// Mitsubishi GX Works2 project: TIMMERs   PLC: Q03UDV

PROGRAM MAIN
VAR
  TS0 : BOOL;
  RT0 : BOOL;
  TMR1 : BOOL;
END_VAR
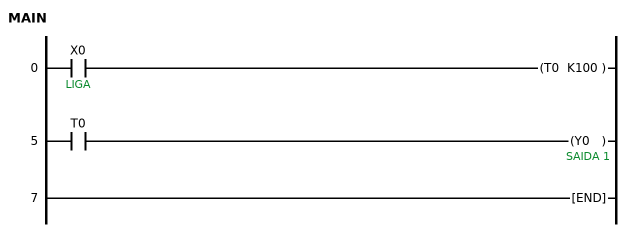
0     LD      X0  ; LIGA
      OUT     T0 K100
5     LD      T0
      OUT     Y0  ; SAIDA 1
7     END
END_PROGRAM

// device comments not shown above
X1  ; DESLIGAR
